{attribute 'strict'}
{attribute 'to_string'}
TYPE
    E_ReleaseState : (
        RELEASE_START      := 0,
        RELEASE_MOVE       := 10,
        RELEASE_MOVE_CHECK := 20,
        RELEASE_FINISHED   := 30,
        RELEASE_ERROR      := 999
    );
END_TYPE

(* stored: Version 1.1.0.1
   DUT E_ReleaseState: Id {a3740f80-971c-438b-aac0-1eb467b77609} *)
